Staubli VAL3: getBitAt.pgx

public program getBitAt(num x_nByteIndex, num x_nBitIndex, num& x_nBuffer[], bool& x_bRes)
  local num l_nResult
  local string l_sByte
  local string l_sMask
  local string l_sResult
begin

  //Header begin

  // This function get the boolean value of the bit number "x_nBitIndex" of the "x_nByteIndex" element (that represent a byte) of the passed array of num (most likely a plc's memory area you read with readArea()).
  //
  //Input parameters
  //
  // num x_nByteIndex: the index of the "x_nBuffer[]" array representing the byte we want to read from (most likely a plc's memory area you read with readArea())
	// num x_nBitIndex: the bit number from 0(LSB) to 7(MSB) in the x_nByteIndex byte, if this value is lower than 0 or higher than 7 x_bRes will be set to false by default.
	// num x_nBuffer[1]: the monodimensional array of num from where we are reading the bit value.
  //
  //Output parameters
  // bool x_bRes: the result, set to "true" if the bit is high, false otherwise.

  //Examples
  //
  // call getBitAt(0,4,l_nRes,l_bRes)
  //
  //History
  // Creation: 24-12-16 - Alessio Villa
  //Header end

  if x_nBitIndex>7
    x_bRes=false
    return
  endIf

  call bitOp:DecToBin(x_nBuffer[x_nByteIndex],l_sByte)
  call bitOp:DecToBin(power(2,x_nBitIndex),l_sMask)
  call bitOp:boolAnd(l_sByte,l_sMask,l_sResult)

  call bitOp:BinToDec(l_sResult,l_nResult)
  if l_nResult>0
    x_bRes=true
  else
    x_bRes=false
  endIf

end
